{attribute 'qualified_only'}
{attribute 'strict'}
TYPE eErrorHandlingSTM :
(
	CheckSystem,
	ShowWarning,
	ShowError,
	Clear
);
END_TYPE

(* stored: Version 1.1.0.1, ProductVersion 3.1.4024.12
   DUT eErrorHandlingSTM: Id {21847fa1-55e7-464a-8c03-3059761eb970} *)
